(* IEC 61131-3 sources: plc_generation_empirical_study/datasets/_archive/native_profile_v4_20260810/tasks/C02_H02_safe_restart_inhibit, 2 files *)

(* ---- interface.st ---- *)
FUNCTION_BLOCK C02_H02_safe_restart_inhibit
VAR_INPUT
    PowerOK : BOOL;
    SafetyOK : BOOL;
    Start : BOOL;
    Stop : BOOL;
    Reset : BOOL;
END_VAR
VAR_OUTPUT
    Running : BOOL;
    RestartInhibit : BOOL;
END_VAR
END_FUNCTION_BLOCK

(* ---- reference.st ---- *)
FUNCTION_BLOCK C02_H02_safe_restart_inhibit
VAR_INPUT
    PowerOK : BOOL;
    SafetyOK : BOOL;
    Start : BOOL;
    Stop : BOOL;
    Reset : BOOL;
END_VAR
VAR_OUTPUT
    Running : BOOL;
    RestartInhibit : BOOL;
END_VAR

IF (NOT PowerOK) OR (NOT SafetyOK) THEN
    Running := FALSE;
    RestartInhibit := TRUE;
ELSIF Stop THEN
    Running := FALSE;
ELSIF Reset AND (NOT Start) THEN
    RestartInhibit := FALSE;
ELSIF Start AND (NOT RestartInhibit) THEN
    Running := TRUE;
END_IF;

IF RestartInhibit THEN
    Running := FALSE;
END_IF;

END_FUNCTION_BLOCK
